(* CODESYS project mqtt-influxdb-codesys-git

Project tree, tasks and I/O mapping:
  Device : CODESYS Control Win V3 x64, 3S - Smart Software Solutions GmbH, version 3.5.16.10
    application Application
      libraries: Standard, * (System); StringUtils, * (System); VisuDialogs, * (System); Web Socket Client SL, 1.9.0.0 (CODESYS); Net Base Services, 3.5.17.0 (3S - Smart Software Solutions GmbH); MQTT Client SL, 1.9.0.0 (CODESYS)
      task MainTask (cyclic, interval t#20ms, priority 1) calls PRG, Pumps_PRG
      task VISU_TASK (cyclic, interval 100 ms, priority 31) calls VisuElems.Visu_Prg
      Funtions/
        function Random [ST]
      global variables GVL
      image pool ImagePool
      text list ModeTextList
      program OEE_PRG [ST]
      program PRG [CFC]
      program PRG [ST]
      program Pumps_PRG [ST]
      text list QoSTextlist
      function TerminateString [ST]
      text list VersionTextList
      visualisation Visualization
    Ethernet : Ethernet, 3S - Smart Software Solutions GmbH, version 3.5.16.0
        settings: IPAddress = [192,168,0,99]; SubnetMask = [255,255,255,0]; GatewayAddress = [0,0,0,0]; NetworkInterfaceName = 'Ethernet 3'; NetworkInterfaceName = "Ethernet 3"; SaveCommunicationSettings = FALSE
      Modbus_TCP_Master : Modbus TCP Master, 3S - Smart Software Solutions GmbH, version 4.3.0.0
          settings: AutoReconnect = TRUE
        Node_Red_Waveshare : Modbus TCP Slave, 3S - Smart Software Solutions GmbH, version 4.1.0.0
            settings: Unit-ID = 1; IPAddress = [127, 0, 0, 1]; Channel 3.Function Code = 15; Channel 3.Read Offset = 0; Channel 3.Read Length = 0; Channel 3.Write Offset = 16#0000; Channel 3.Write Length = 8; Channel 3.Cycle Time = 100
            output Application.Pumps_PRG.byPumps : BYTE  // Channel 3.Channel 3
            unmapped channels: Channel 3
  libraries: VisuSymbols, 4.4.0.0 (System)
  5ce3da45-db07-42e7-a21c-a00fff4ed8f6|C:\Users\a.werner\Documents\background.jpg
  text list GlobalTextList
*)

// Device/Application/GVL
//{attribute 'qualified_only'}
VAR_GLOBAL
	 Seed : UDINT := 123456789; // Initial seed (should be changed)
END_VAR

// Device/Application/PRG
// MQTT Client with visualization
PROGRAM PRG
VAR
	mqttClient : MQTT.MQTTClient; // Function block to establish a connection to a MQTT broker
	mqttPublisher : MQTT.MQTTPublish; // Function block to publish MQTT messages
	mqttPublisher2 : MQTT.MQTTPublish; // Function block to publish MQTT messages
	mqttSubscriber : MQTT.MQTTSubscribe; // Function block to subscribe MQTT topics
	mqttSubscriber2 : MQTT.MQTTSubscribe; // Function block to subscribe MQTT topics
	sHostname : STRING(255) := ''; // Hostname or ip address or URL (for WebSockets: ws:// or wss://)
	uiPort : UINT := 1883; // Port of the MQTT broker
	wsPublishTopic : WSTRING(1024) := ""; // Topic to publish a message
	wsPublishTopic2 : WSTRING(1024) := ""; // Topic to publish a message
	wsSubcribeTopicFilter : WSTRING(1024) := ""; // Topic filter to subcribe a topic
	wsSubcribeTopicFilter2 : WSTRING(1024) := ""; // Topic filter to subcribe a topic
	sWillMessage : STRING(1024); // The last will message
	sPublishMessage : STRING(1024) := ''; // The messsage to publish
	sPublishMessage2 : STRING(1024) := ''; // The messsage to publish
	sSubscribeMessage : STRING(4096); // Message buffer with the retrieved message  
	sSubscribeMessage2 : STRING(4096); // Message buffer with the retrieved message  
	rsPub1Error: RS; // Helper to publisher state
	rsPub1Done: RS; // Helper to publisher state
	rsPub2Error: RS; // Helper to publisher state
	rsPub2Done: RS; // Helper to publisher state
	eCommunicationMode : MQTT.COMMUNICATION_MODE := MQTT.COMMUNICATION_MODE.TCP; // Communication mode: TCP/IP or WebSockets
	eMQTTVersion : MQTT.MQTT_VERSION := MQTT.MQTT_VERSION.V3_1_1; // The MQTT protocol version

	// Example of connect properties (V5 only)
	mQTTConnectProperties : MQTT.MQTTConnectProperties := (
		udiSessionExpiryInterval := 10,
		udiMaximumPacketSize := MQTT.MQTTParam.g_udiMaxPacketSize,
		userProperties := 
			[
				(wsKey := "key1", wsValue := "value1"),
				(wsKey := "key2", wsValue := "value2"),	
				(wsKey := "key3", wsValue := "value3")
			]
	);
	
	// Example of will properties (V5 only)
	mQTTWillProperties : MQTT.MQTTWillProperties := (
		bPayloadFormatIndicator := 1, // 1: UTF-8, 0: Binary
		wsContentType := "text/plain",
		udiMessageExpiryInterval := 60,
		udiWillDelayInterval := 60,
		userProperties := 
		[
			(wsKey := "key1", wsValue := "value1"),
		 	(wsKey := "key2", wsValue := "value2"),	
			(wsKey := "key3", wsValue := "value3")
		]);
	
	// Example of publish properties (V5 only)
	mqTTPublishProperties : MQTT.MQTTPublishProperties := (
		bPayloadFormatIndicator := 1, // 1: UTF-8, 0: Binary
		wsContentType := "text/plain",
		udiMessageExpiryInterval := 60,
		userProperties := 
		[
			(wsKey := "key1", wsValue := "value1"),
		 	(wsKey := "key2", wsValue := "value2"),	
			(wsKey := "key3", wsValue := "value3")
		]
	);
	
	// Example of subscribe properties (V5 only)
	mQTTSubscribeProperties : MQTT.MQTTSubscribeProperties := (
		udiSubscriptionIdentifier := 4343,
		userProperties := 
		[
			(wsKey := "key1", wsValue := "value1"),
		 	(wsKey := "key2", wsValue := "value2"),	
			(wsKey := "key3", wsValue := "value3")
		],
		xNoLocalOption := FALSE
	);
	
	/// If you want to use client certificates, you can configure the connection via the TLS context.
	//
	// Example (static):
	//
	// _sCommonName : STRING := 'COMMON_NAME_OF_CERTIFICATE'; // CN of the certificate (common name). 
	// _sCipherList : NBS.CIPHER_LIST := STRUCT(psList := ADR('HIGH'), udiSize := 5); // Cipher string see https://www.openssl.org/docs/man1.1.1/man1/ciphers.html
	// _ciDefaultCertInfo : NBS.CERT_INFO := (psInfo := ADR(_sCommonName), udiSize := SIZEOF(_sCommonName)); // CN of the certificate (common name)
	
	// _tlsContext : NBS.TLSContext := (	sUseCaseName := _sCommonName, // A certificate is stored in the certificate store with the use case name. You can choose any name. Here we use the common name.
	//									ePurpose := NBS.PURPOSE.CLIENT_SIDE, // For client certificates set this to NBS.PURPOSE.CLIENT_SIDE
	//									sTLSVersion := '1.2', // The TLS version
	//									sCipherList := _sCipherList, // Set the cipher list
	//									sHostname := 'HOSTNAME_OF_THE_BROKER', // The hostname of the broker
	//									udiVerificationMode := 2, // 2 => Active Peer verification
	//									ciCertInfo := _ciDefaultCertInfo, // Set the cert info
	//									itfCertVerifer := 0); // 0 => No Verifier 
	// 
	// mqttClient : MQTT.MQTTClient := (itfTLSCOntext := _tlsContext);
    //
	// You can use the method TLSContext.SetInitialValue to set the context while runtime and set the context via the input itfTLSCOntext of the client FB.
END_VAR

// Connect to a MQTT broker
mqttClient(
    uiPort := uiPort,
    pbWillMessage := ADR(sWillMessage),
    uiWillMessageSize := DINT_TO_UINT(Stu.StrLenA(ADR(sWillMessage))),
    eCommunicationMode := eCommunicationMode,
    sWebSocketUrl := sHostname,
    eMQTTVersion := eMQTTVersion,
    mQTTConnectProperties := mQTTConnectProperties,
    mQTTWillProperties := mQTTWillProperties,
    sHostname := sHostname); // MQTT.MQTTClient
// Subscribe a topic
mqttSubscriber(
    pbPayload := ADR(sSubscribeMessage),
    udiMaxPayloadSize := SIZEOF(sSubscribeMessage),
    mQTTSubscribeProperties := mQTTSubscribeProperties,
    mqttClient := mqttClient,
    wsTopicFilter := wsSubcribeTopicFilter); // MQTT.MQTTSubscribe
TerminateString(psIn := ADR(sSubscribeMessage), udiLength := mqttSubscriber.udiPayloadSize);
// Subscribe a second topic
mqttSubscriber2(
    pbPayload := ADR(sSubscribeMessage2),
    udiMaxPayloadSize := SIZEOF(sSubscribeMessage2),
    mqttClient := mqttClient,
    wsTopicFilter := wsSubcribeTopicFilter2); // MQTT.MQTTSubscribe
TerminateString(psIn := ADR(sSubscribeMessage2), udiLength := mqttSubscriber2.udiPayloadSize);
// Pulish a message
mqttPublisher(
    udiTimeOut := 10000000,
    pbPayload := ADR(sPublishMessage),
    udiPayloadSize := DINT_TO_UDINT(Stu.StrLenA(ADR(sPublishMessage))),
    mQTTPublishProperties := mqTTPublishProperties,
    mqttClient := mqttClient,
    wsTopicName := wsPublishTopic); // MQTT.MQTTPublish
rsPub1Done(SET := mqttPublisher.xDone, RESET1 := mqttPublisher.xBusy); // RS
rsPub1Error(SET := mqttPublisher.xError, RESET1 := mqttPublisher.xBusy); // RS
// Pulish a second message
mqttPublisher2(
    udiTimeOut := 10000000,
    pbPayload := ADR(sPublishMessage2),
    udiPayloadSize := DINT_TO_UDINT(Stu.StrLenA(ADR(sPublishMessage2))),
    mqttClient := mqttClient,
    wsTopicName := wsPublishTopic2); // MQTT.MQTTPublish
rsPub2Done(SET := mqttPublisher2.xDone, RESET1 := mqttPublisher2.xBusy); // RS
rsPub2Error(SET := mqttPublisher2.xError, RESET1 := mqttPublisher2.xBusy); // RS

END_PROGRAM

// Device/Application/TerminateString
// Terminates the STRING psIn at position udiLength
FUNCTION TerminateString : BOOL
VAR_INPUT
	psIn : POINTER TO BYTE; // Pointer to STRING
	udiLength : UDINT; // Length of psIn
END_VAR
VAR
END_VAR

psIn[udiLength] := 0;
TerminateString := TRUE;

END_FUNCTION

// Device/Application/PRG
PROGRAM PRG
VAR

	mqttClient : MQTT.MQTTClient; // Function block to establish a connection to a MQTT broker
	mqttPublisher : MQTT.MQTTPublish; // Function block to publish MQTT messages
	mqttPublisher2 : MQTT.MQTTPublish; // Function block to publish MQTT messages
	mqttSubscriber : MQTT.MQTTSubscribe; // Function block to subscribe MQTT topics
	mqttSubscriber2 : MQTT.MQTTSubscribe; // Function block to subscribe MQTT topics
	sHostname : STRING(255) := ''; // Hostname or ip address or URL (for WebSockets: ws:// or wss://)
	uiPort : UINT := 1883; // Port of the MQTT broker
	wsPublishTopic : WSTRING(1024) := ""; // Topic to publish a message
	wsPublishTopic2 : WSTRING(1024) := ""; // Topic to publish a message
	wsSubcribeTopicFilter : WSTRING(1024) := ""; // Topic filter to subcribe a topic
	wsSubcribeTopicFilter2 : WSTRING(1024) := ""; // Topic filter to subcribe a topic
	sWillMessage : STRING(1024); // The last will message
	sPublishMessage : WSTRING(1024); // The messsage to publish
	sPublishMessage2 : STRING(1024) := ''; // The messsage to publish
	sSubscribeMessage : STRING(4096); // Message buffer with the retrieved message  
	sSubscribeMessage2 : STRING(4096); // Message buffer with the retrieved message  
	rsPub1Error: RS; // Helper to publisher state
	rsPub1Done: RS; // Helper to publisher state
	rsPub2Error: RS; // Helper to publisher state
	rsPub2Done: RS; // Helper to publisher state
	eCommunicationMode : MQTT.COMMUNICATION_MODE := MQTT.COMMUNICATION_MODE.TCP; // Communication mode: TCP/IP or WebSockets
	eMQTTVersion : MQTT.MQTT_VERSION := MQTT.MQTT_VERSION.V3_1_1; // The MQTT protocol version
	udiLength : UDINT;
	// Example of connect properties (V5 only)
	mQTTConnectProperties : MQTT.MQTTConnectProperties := (
		udiSessionExpiryInterval := 10,
		udiMaximumPacketSize := MQTT.MQTTParam.g_udiMaxPacketSize,
		userProperties := 
			[
				(wsKey := "key1", wsValue := "value1"),
				(wsKey := "key2", wsValue := "value2"),	
				(wsKey := "key3", wsValue := "value3")
			]
	);
	
	// Example of will properties (V5 only)
	mQTTWillProperties : MQTT.MQTTWillProperties := (
		bPayloadFormatIndicator := 1, // 1: UTF-8, 0: Binary
		wsContentType := "text/plain",
		udiMessageExpiryInterval := 60,
		udiWillDelayInterval := 60,
		userProperties := 
		[
			(wsKey := "key1", wsValue := "value1"),
		 	(wsKey := "key2", wsValue := "value2"),	
			(wsKey := "key3", wsValue := "value3")
		]);
	
	// Example of publish properties (V5 only)
	mqTTPublishProperties : MQTT.MQTTPublishProperties := (
		bPayloadFormatIndicator := 1, // 1: UTF-8, 0: Binary
		wsContentType := "text/plain",
		udiMessageExpiryInterval := 60,
		userProperties := 
		[
			(wsKey := "key1", wsValue := "value1"),
		 	(wsKey := "key2", wsValue := "value2"),	
			(wsKey := "key3", wsValue := "value3")
		]
	);
	
	// Example of subscribe properties (V5 only)
	mQTTSubscribeProperties : MQTT.MQTTSubscribeProperties := (
		udiSubscriptionIdentifier := 4343,
		userProperties := 
		[
			(wsKey := "key1", wsValue := "value1"),
		 	(wsKey := "key2", wsValue := "value2"),	
			(wsKey := "key3", wsValue := "value3")
		],
		xNoLocalOption := FALSE
	);
	
	/// If you want to use client certificates, you can configure the connection via the TLS context.
	//
	// Example (static):
	//
	// _sCommonName : STRING := 'COMMON_NAME_OF_CERTIFICATE'; // CN of the certificate (common name). 
	// _sCipherList : NBS.CIPHER_LIST := STRUCT(psList := ADR('HIGH'), udiSize := 5); // Cipher string see https://www.openssl.org/docs/man1.1.1/man1/ciphers.html
	// _ciDefaultCertInfo : NBS.CERT_INFO := (psInfo := ADR(_sCommonName), udiSize := SIZEOF(_sCommonName)); // CN of the certificate (common name)
	
	// _tlsContext : NBS.TLSContext := (	sUseCaseName := _sCommonName, // A certificate is stored in the certificate store with the use case name. You can choose any name. Here we use the common name.
	//									ePurpose := NBS.PURPOSE.CLIENT_SIDE, // For client certificates set this to NBS.PURPOSE.CLIENT_SIDE
	//									sTLSVersion := '1.2', // The TLS version
	//									sCipherList := _sCipherList, // Set the cipher list
	//									sHostname := 'HOSTNAME_OF_THE_BROKER', // The hostname of the broker
	//									udiVerificationMode := 2, // 2 => Active Peer verification
	//									ciCertInfo := _ciDefaultCertInfo, // Set the cert info
	//									itfCertVerifer := 0); // 0 => No Verifier 
	// 
	// mqttClient : MQTT.MQTTClient := (itfTLSCOntext := _tlsContext);
    //
	// You can use the method TLSContext.SetInitialValue to set the context while runtime and set the context via the input itfTLSCOntext of the client FB.
END_VAR

mqttClient(
	xEnable:= , 
	xDone=> , 
	xBusy=> , 
	xError=> , 
	uiPort:= uiPort, 
	xUseTLS:= , 
	uiKeepAlive:= , 
	pbWillMessage:= ADR(sWillMessage), 
	uiWillMessageSize:= DINT_TO_UINT(Stu.StrLenA(ADR(sWillMessage))), 
	xWillRetain:= , 
	eWillQoS:= , 
	xCleanSession:= , 
	wsUsername:= , 
	wsPassword:= , 
	wsWillTopic:= , 
	sClientId:= , 
	tPingInterval:= , 
	hCert:= , 
	itfTLSContext:= , 
	itfAsyncProperty:= , 
	udiTimeOut:= , 
	eCommunicationMode:= eCommunicationMode, 
	sWebSocketUrl:= sHostname, 
	eMQTTVersion:= eMQTTVersion, 
	mQTTConnectProperties:= mQTTConnectProperties, 
	mQTTWillProperties:= mQTTWillProperties, 
	sHostname:= sHostname, 
	eMQTTError=> , 
	xConnectedToBroker=> , 
	eReaonCode=> , 
	mQTTConnackProperties=> );
	
	// subscribe to a topic subscriber 1
	mqttSubscriber(
	xEnable:= , 
	xDone=> , 
	xBusy=> , 
	xError=> , 
	eSubscribeQoS:= , 
	pbPayload:= ADR(sSubscribeMessage), 
	udiMaxPayloadSize:= SIZEOF(sSubscribeMessage), 
	eFilterMode:= , 
	mQTTSubscribeProperties:= mQTTSubscribeProperties, 
	udiTimeout:= , 
	mqttClient:= mqttClient, 
	wsTopicFilter:= wsSubcribeTopicFilter, 
	eMQTTError=> , 
	xReceived=> , 
	udiPayloadSize=> , 
	xSubscribeActive=> , 
	wsLastTopic=> , 
	mQTTPublishProperties=> );
	
	TerminateString(psIn:= ADR(sSubscribeMessage), udiLength:= mqttSubscriber.udiMaxPayloadSize );

// subscribe to a topic subscriber 1
mqttSubscriber2(
	xEnable:= , 
	xDone=> , 
	xBusy=> , 
	xError=> , 
	eSubscribeQoS:= , 
	pbPayload:= ADR(sSubscribeMessage2), 
	udiMaxPayloadSize:= SIZEOF(sSubscribeMessage2), 
	eFilterMode:= , 
	mQTTSubscribeProperties:= mQTTSubscribeProperties, 
	udiTimeout:= , 
	mqttClient:= mqttClient, 
	wsTopicFilter:= wsSubcribeTopicFilter2, 
	eMQTTError=> , 
	xReceived=> , 
	udiPayloadSize=> , 
	xSubscribeActive=> , 
	wsLastTopic=> , 
	mQTTPublishProperties=> );
	
	TerminateString(psIn:= ADR(sSubscribeMessage2), udiLength:= mqttSubscriber2.udiMaxPayloadSize );

// Publish a message 1
//sPublishMessage := TO_STRING(OEE_PRG.OEE);
sPublishMessage := OEE_PRG.wsJsonData;
udiLength:=Stu.StrLenW(ADR(sPublishMessage))*2;
	
mqttPublisher(
	xExecute:= , 
	udiTimeOut:= 10000000, 
	xDone=> , 
	xBusy=> , 
	xError=> , 
	eQoS:= , 
	xReDelivery:= , 
	xRetain:= , 
	pbPayload:= ADR(sPublishMessage), 
	udiPayloadSize:= udiLength, 
	mQTTPublishProperties:= mqTTPublishProperties, 
	mqttClient:= mqttClient, 
	wsTopicName:= wsPublishTopic, 
	eMQTTError=> );
	
rsPub1Done(
	SET:= mqttPublisher.xDone,
	RESET1:= mqttPublisher.xBusy,
);

rsPub1Error(
	SET:= mqttPublisher.xError,
	RESET1:= mqttPublisher.xBusy  );
	
// Publish a message 2
mqttPublisher2(
    xExecute:= ,
    udiTimeOut:= 10000000,
    xDone=> ,
    xBusy=> ,
    xError=> ,
    eQoS:= ,
    xReDelivery:= ,
    xRetain:= ,
    pbPayload:= ADR(sPublishMessage2),
    udiPayloadSize:= DINT_TO_UDINT(Stu.StrLenA(ADR(sPublishMessage2))),
    mQTTPublishProperties:= mqTTPublishProperties,
    mqttClient:= mqttClient,
    wsTopicName:= wsPublishTopic2,
    eMQTTError=> );
	
rsPub2Done(
    SET:= mqttPublisher2.xDone,
    RESET1:= mqttPublisher2.xBusy
);

rsPub2Error(
    SET:= mqttPublisher2.xError,
    RESET1:= mqttPublisher2.xBusy
);

END_PROGRAM

// Device/Application/OEE_PRG
PROGRAM OEE_PRG
VAR
    // MQTT Client configuration
    mqttClient : MQTT.MQTTClient;
    MQTT_Payload : STRING(255);

    // Production data
    OEE : REAL := 50.0; // Overall Equipment Effectiveness
    Performance : REAL := 75.0; // Machine performance percentage
    Quality : REAL := 80.0; // Quality percentage
    Availability : REAL := 95.0; // Machine availability percentage
    
    MachineState : STRING(20) := 'Running'; // Machine status
    GoodParts : INT := 0; // Number of good parts produced
    BadParts : INT := 0; // Number of defective parts
    ProductWeight : REAL := 5040.0; // Weight of the product

    // Timer for data updates
    Timer : TON;
END_VAR

//MQTT Client Configuration
mqttClient.sHostname := '192.168.10.16'; // MQTT Broker IP
mqttClient.uiPort := 1883; // Default MQTT port
mqttClient.sClientID := 'CodesysClient';
// mqttClient.wsUsername := 'mqtt_user'; // Optional - set if authentication is required
// mqttClient.wsPassword := 'mqtt_password'; // Optional - set if authentication is required
// mqttClient.wsWillTopic := 'factory/status'; // Will topic if the connection is lost
mqttClient.pbWillMessage := ADR('{"status":"offline"}'); // Will message payload
mqttClient.uiWillMessageSize := DINT_TO_UINT(Stu.StrLenA(ADR('{"status":"offline"}')));
mqttClient.xWillRetain := FALSE;
mqttClient.eWillQoS := MQTT.QOS.QOS1;
mqttClient.xCleanSession := TRUE;
// mqttClient.sTopic := 'factory/data';
mqttClient.uiKeepAlive := 60;
mqttClient.xEnable := TRUE;

// Data update every 5 seconds
Timer(IN := TRUE, PT := T#5S);

// Random data generation for OEE and production metrics
IF Timer.Q THEN
    OEE := 50.0 + REAL(RANDOM() * 20.0); // Simulate OEE fluctuation
    Performance := 70.0 + REAL(RANDOM() * 10.0); // Performance percentage
    Quality := 75.0 + REAL(RANDOM() * 10.0); // Quality percentage
    Availability := 90.0 + REAL(RANDOM() * 10.0); // Machine uptime percentage

    // Simulating machine state: Running or Stopped
    IF RANDOM() > 0.5 THEN
        MachineState := 'Stopped';
    ELSE
        MachineState := 'Running';
    END_IF;

    // Production part counts
    GoodParts := GoodParts + 1 + INT(RANDOM() * 3); // Increment good parts
    BadParts := BadParts + INT(RANDOM() * 2); // Increment defective parts

    // Simulate product weight variations
    ProductWeight := 5040.0 + RANDOM() * 50.0;

    // Format data in JSON format for MQTT transmission
    MQTT_Payload := CONCAT(
        '{"OEE":', REAL_TO_STRING(OEE), 
        ',"Performance":', REAL_TO_STRING(Performance),
        ',"Quality":', REAL_TO_STRING(Quality),
        ',"Availability":', REAL_TO_STRING(Availability),
        ',"MachineState":"', MachineState, '"',
        ',"GoodParts":', INT_TO_STRING(GoodParts),
        ',"BadParts":', INT_TO_STRING(BadParts),
        ',"ProductWeight":', REAL_TO_STRING(ProductWeight),
        '}'
    );

    // Send JSON data to MQTT topic
    mqttClient.PublishMessage('factory/data', MQTT_Payload, MQTT.QOS.QOS1, FALSE);

    // Restart timer for next update
    Timer(IN := FALSE);
    Timer(IN := TRUE);
END_IF

END_PROGRAM

// Device/Application/Funtions/Random
FUNCTION Random : REAL
VAR_INPUT
END_VAR

VAR CONSTANT
    A : UDINT := 1664525;      // Multiplier
    C : UDINT := 1013904223;   // Increment
    M : REAL := 4294967296;   // Modulus (2^32)
END_VAR

VAR
    RandomValue : UDINT;
END_VAR

// Update seed using LCG formula
Seed := (A * Seed + C) MOD UDINT#4294967295; // Correct modulus for UDINT

// Convert result to REAL in range 0.0 - 1.0
Random := UDINT_TO_REAL(Seed) / UDINT_TO_REAL(M);

END_FUNCTION

// Device/Application/Pumps_PRG
PROGRAM Pumps_PRG
VAR
	byPumps: byte;
	
	byTest: BYTE;
END_VAR

// Pump nr 1
IF PRG.wsPublishTopic = "factory/pumpstation/pump1" AND PRG.sSubscribeMessage = TO_STRING("ON") THEN
    byPumps.0 := TRUE;
ELSIF PRG.wsPublishTopic = "factory/pumpstation/pump1" AND PRG.sSubscribeMessage = TO_STRING("OFF") THEN
    byPumps.0 := FALSE;
END_IF

// Pump nr 2
IF PRG.wsPublishTopic = "factory/pumpstation/pump2" AND PRG.sSubscribeMessage = TO_STRING("START") THEN
    byPumps.1 := TRUE;
ELSIF PRG.wsPublishTopic = "factory/pumpstation/pump2" AND PRG.sSubscribeMessage = TO_STRING("OFF") THEN
    byPumps.1 := FALSE;
END_IF

// Pump nr 3
IF PRG.wsPublishTopic = "factory/pumpstation/pump3" AND PRG.sSubscribeMessage = TO_STRING("ENABLE") THEN
    byPumps.2 := TRUE;
ELSIF PRG.wsPublishTopic = "factory/pumpstation/pump3" AND PRG.sSubscribeMessage = TO_STRING("OFF") THEN
    byPumps.2 := FALSE;
END_IF

END_PROGRAM

// Device/Application/Visualization
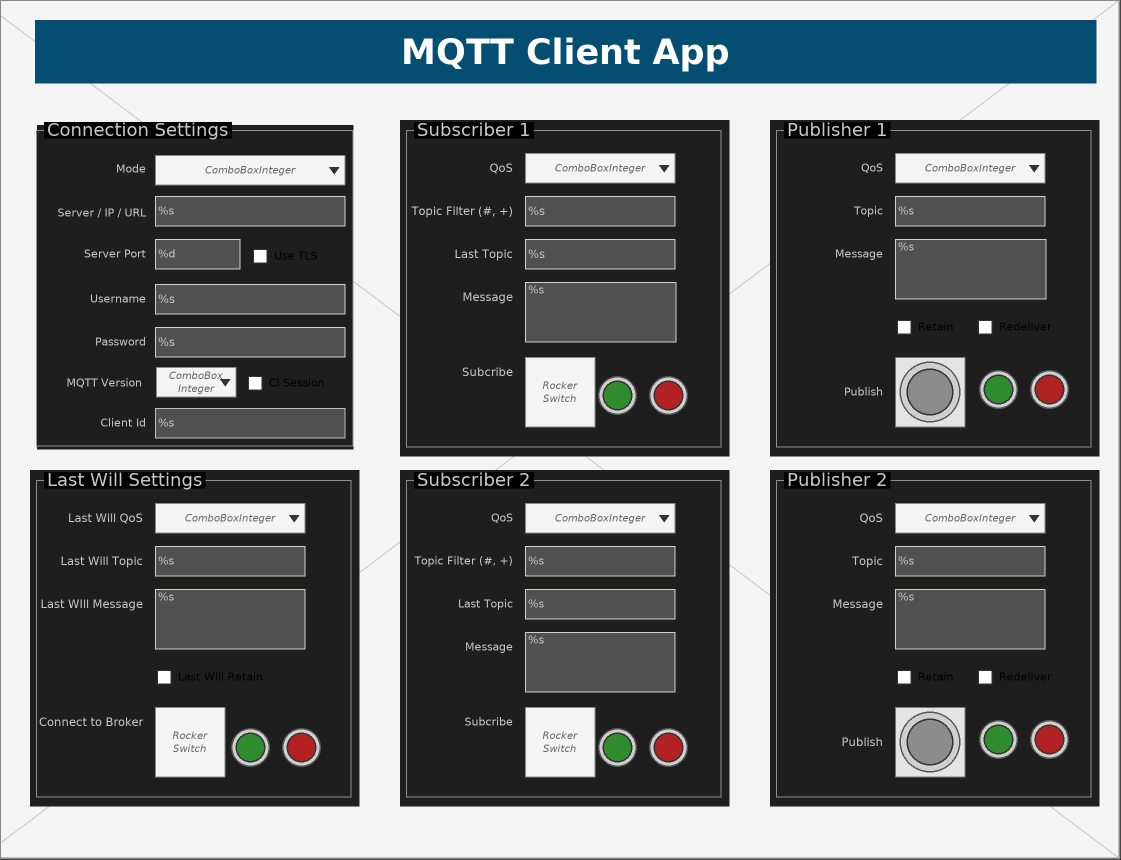
VISUALIZATION Visualization  // 1121x860
    Image (-20,0 1139x858), image: ImagePool.background
    Rectangle (37,125 316x324)
    Rectangle (30,470 329x336)
    GroupBox (36,472 315x325), "Last Will Settings"
        ComboBoxInteger (119,31 150x30), variable: PRG.mqttClient.eWillQoS, text list: 'QoSTextlist'
        Lamp1 (192,253 45x45), variable: PRG.mqttClient.xConnectedToBroker, style: Lamp-Lamp1-Green
        Lamp1 (243,253 45x45), variable: PRG.mqttClient.xError, style: Lamp-Lamp1-Red
    Label (46,503 100x30), "Last Will QoS"
    Textfield (155,546 150x30), "%s", text variable: PRG.mqttClient.wsWillTopic
        OnMouseClick: write the text variable via Default
    Label (46,546 100x30), "Last Will Topic"
    Textfield (155,589 150x60), "%s", text variable: PRG.sWillMessage
        OnMouseClick: write the text variable via Default
    Label (46,589 100x30), "Last WIll Message"
    Checkbox (155,662 150x30), "Last Will Retain", variable: PRG.mqttClient.xWillRetain
    Label (46,707 100x30), "Connect to Broker"
    RockerSwitch (155,707 70x70), variable: PRG.mqttClient.xEnable, behaviour: TOGGLE, style: Switch-RockerSwitch-Gray
    Group (770,120 329x336)
        Rectangle (0,0 329x336)
        GroupBox (6,2 315x325), "Publisher 1"
        ComboBoxInteger (125,33 150x30), variable: PRG.mqttPublisher.eQoS, text list: 'QoSTextlist'
        Label (16,33 100x30), "QoS"
        Textfield (125,76 150x30), "%s", text variable: PRG.wsPublishTopic
            OnMouseClick: write the text variable via Default
        Label (16,76 100x30), "Topic"
        Textfield (125,119 151x60), "%s", text variable: PRG.sPublishMessage
            OnMouseClick: write the text variable via Default
        Label (16,119 100x30), "Message"
        Checkbox (125,192 79x30), "Retain", variable: PRG.mqttPublisher.xRetain
        Checkbox (206,192 97x30), "Redeliver", variable: PRG.mqttPublisher.xReDelivery
        PushSwitch (125,237 70x70), variable: PRG.mqttPublisher.xExecute, input disabled if: NOT PRG.mqttClient.xConnectedToBroker, behaviour: TAP, style: Switch-PushSwitch-Gray
        Label (16,257 100x30), "Publish"
        Lamp1 (206,247 45x45), variable: PRG.rsPub1Done.Q1, style: Lamp-Lamp1-Green
        Lamp1 (257,247 45x45), variable: PRG.rsPub1Error.Q1, style: Lamp-Lamp1-Red
    Rectangle (770,470 329x336)
    GroupBox (776,472 315x325), "Publisher 2"
    ComboBoxInteger (895,503 150x30), variable: PRG.mqttPublisher2.eQoS, text list: 'QoSTextlist'
    Label (786,503 100x30), "QoS"
    Textfield (895,546 150x30), "%s", text variable: PRG.wsPublishTopic2
        OnMouseClick: write the text variable via Default
    Label (786,546 100x30), "Topic"
    Textfield (895,589 150x60), "%s", text variable: PRG.sPublishMessage2
        OnMouseClick: write the text variable via Default
    Label (786,589 100x30), "Message"
    Checkbox (895,662 80x30), "Retain", variable: PRG.mqttPublisher2.xRetain
    Checkbox (976,662 96x30), "Redeliver", variable: PRG.mqttPublisher2.xReDelivery
    PushSwitch (895,707 70x70), variable: PRG.mqttPublisher2.xExecute, input disabled if: NOT PRG.mqttClient.xConnectedToBroker, behaviour: TAP, style: Switch-PushSwitch-Gray
    Label (786,727 100x30), "Publish"
    Lamp1 (976,717 45x45), variable: PRG.rsPub2Done.Q1, style: Lamp-Lamp1-Green
    Lamp1 (1027,717 45x45), variable: PRG.rsPub2Error.Q1, style: Lamp-Lamp1-Red
    Rectangle (400,470 329x336)
    GroupBox (406,472 315x325), "Subscriber 2"
        Lamp1 (189,253 45x45), variable: PRG.mqttSubscriber2.xSubscribeActive, style: Lamp-Lamp1-Green
        Lamp1 (240,253 45x45), variable: PRG.mqttSubscriber2.xError, style: Lamp-Lamp1-Red
    ComboBoxInteger (525,503 150x30), variable: PRG.mqttSubscriber2.eSubscribeQoS, text list: 'QoSTextlist'
    Label (416,503 100x30), "QoS"
    Textfield (525,546 150x30), "%s", text variable: PRG.wsSubcribeTopicFilter2
        OnMouseClick: write the text variable via Default
    Label (416,546 100x30), "Topic Filter (#, +)"
    Textfield (525,632 150x60), "%s", text variable: PRG.sSubscribeMessage2
    Label (416,632 100x30), "Message"
    RockerSwitch (525,707 70x70), variable: PRG.mqttSubscriber2.xEnable, input disabled if: NOT PRG.mqttClient.xConnectedToBroker, behaviour: TOGGLE, style: Switch-RockerSwitch-Gray
    Label (416,707 100x30), "Subcribe"
    Label (416,589 100x30), "Last Topic"
    Textfield (525,589 150x30), "%s", text variable: PRG.mqttSubscriber2.wsLastTopic
    Rectangle (400,120 329x336)
    GroupBox (406,122 315x325), "Subscriber 1"
        Lamp1 (189,251 45x45), variable: PRG.mqttSubscriber.xSubscribeActive, style: Lamp-Lamp1-Green
        Lamp1 (240,251 45x45), variable: PRG.mqttSubscriber.xError, style: Lamp-Lamp1-Red
    ComboBoxInteger (525,153 150x30), variable: PRG.mqttSubscriber.eSubscribeQoS, text list: 'QoSTextlist'
    Label (416,153 100x30), "QoS"
    Textfield (525,196 150x30), "%s", text variable: PRG.wsSubcribeTopicFilter
        OnMouseClick: write the text variable via Default
    Label (416,196 100x30), "Topic Filter (#, +)"
    Textfield (525,282 151x60), "%s", text variable: PRG.sSubscribeMessage
    Label (416,282 100x30), "Message"
    RockerSwitch (525,357 70x70), variable: PRG.mqttSubscriber.xEnable, input disabled if: NOT PRG.mqttClient.xConnectedToBroker, behaviour: TOGGLE, style: Switch-RockerSwitch-Gray
    Label (416,357 100x30), "Subcribe"
    Label (416,239 100x30), "Last Topic"
    Textfield (525,239 150x30), "%s", text variable: PRG.mqttSubscriber.wsLastTopic
    GroupBox (36,122 317x324), "Connection Settings"
        ComboBoxInteger (119,33 190x30), variable: PRG.eCommunicationMode, text list: 'ModeTextList'
        Label (-23,32 136x30), "Mode"
        Textfield (119,74 190x30), "%s", text variable: PRG.sHostname
            OnMouseClick: write the text variable via Default
        Label (13,117 100x30), "Server Port", invisible if: PRG.eCommunicationMode = MQTT.COMMUNICATION_MODE.WEB_SOCKET
        Label (13,286 100x30), "Client Id"
        Textfield (119,286 190x30), "%s", text variable: PRG.mqttClient.sClientId
            OnMouseClick: write the text variable via Default
        Label (13,205 100x30), "Password"
        Textfield (119,205 190x30), "%s", text variable: PRG.mqttClient.wsPassword
            OnMouseClick: write the text variable via Default
        Label (13,162 100x30), "Username"
        Textfield (119,162 190x30), "%s", text variable: PRG.mqttClient.wsUsername
            OnMouseClick: write the text variable via Default
        Textfield (119,117 85x30), "%d", text variable: PRG.uiPort, invisible if: PRG.eCommunicationMode = MQTT.COMMUNICATION_MODE.WEB_SOCKET
            OnMouseClick: write the text variable via Default
        Label (-12,76 125x30), "Server / IP / URL"
        Checkbox (215,119 75x30), "Use TLS", variable: PRG.mqttClient.xUseTLS, invisible if: PRG.eCommunicationMode = MQTT.COMMUNICATION_MODE.WEB_SOCKET
        ComboBoxInteger (120,245 80x30), variable: PRG.eMQTTVersion, text list: 'VersionTextList'
        Label (23,246 86x30), "MQTT Version"
        Checkbox (210,246 103x30), "Cl Session", variable: PRG.mqttClient.xCleanSession
    Rectangle (35,20 1061x63), "MQTT Client App"
END_VISUALIZATION

(* text list ModeTextList (id | default)
  0 | TCP/IP
  1 | WebSocket
   |  *)

(* text list QoSTextlist (id | default)
  0 | QoS 0
  1 | QoS 1
  2 | QoS 2
   |  *)

(* text list VersionTextList (id | default)
  0 | 3.1.1
  1 | 5.0
   |  *)
